TYPE ST_WeighingStaton_Settings :
STRUCT
END_STRUCT
END_TYPE

(* stored: Version 1.1.0.1, ProductVersion 3.1.4024.15
   DUT ST_WeighingStaton_Settings: Id {d0ad0e00-53b8-4ef3-adb4-b919773c252b} *)
